// TIA Portal V17 export
// export: Created 2024-09-27T18:55:49.6572853Z, ExportSetting WithDefaults, DisplayName Totally Integrated Automation Portal, DisplayVersion V17, DisplayName TIA Portal Openness, DisplayVersion V17, DisplayName TIA Portal Version Control Interface, DisplayVersion V17, DisplayName STEP 7 Professional, DisplayVersion V17, DisplayName STEP 7 Safety, DisplayVersion V17, DisplayName WinCC Professional, DisplayVersion V17
DATA_BLOCK "proces_value"   // DB12
{ S7_Optimized_Access := 'TRUE' }
VERSION : 0.1
// stored: AutoNumber true, DBAccessibleFromOPCUA true, IsOnlyStoredInLoadMemory false, IsRetainMemResEnabled false, IsWriteProtectedInAS false, MemoryReserve 100
   VAR RETAIN
      db_tp_akt_pred_stołu : Real := 50.0;
   END_VAR
   VAR
      db_tp_nowa_pred_stołu : Real;
   END_VAR
   VAR RETAIN
      db_tp_akt_takt_stołu : Time := T#7S;
   END_VAR
   VAR
      db_tp_nowy_takt_stołu : Real;
   END_VAR
   VAR RETAIN
      db_tp_akt_czas_ssania : Time := T#1S;
   END_VAR
   VAR
      db_tp_nowy_czas_ssania : Real;
   END_VAR
   VAR RETAIN
      "db_tp_akt_czas przedmuchu" : Time := T#1S;
   END_VAR
   VAR
      db_tp_nowy_czas_przedmuchu : Real;
   END_VAR
   VAR RETAIN
      db_tp_akt_delay_sił_zag : Time := T#100MS;
   END_VAR
   VAR
      db_tp_nowy_delay_sił_zag : Real;
   END_VAR
   VAR RETAIN
      db_tp_akt_delay_sił_odbioru_stoł : Time := T#1S;
   END_VAR
   VAR
      db_tp_nowy_delay_sił_odbioru_stoł : Real;
   END_VAR
   VAR RETAIN
      db_licznik_calkowity : DInt;
      db_licznik_zadane : DInt;
      db_licznik_wykonane : DInt;
      db_aktualne_gniazdo : Int;
      db_auto_table_velocity : Real := 0.5;
   END_VAR
BEGIN
END_DATA_BLOCK
